// Brief: Setup Arm Error Hold
FUNCTION_BLOCK PUBLIC FB_SetupCtrlError EXTENDS FB_SetupArmCtrlBase
VAR_INPUT
END_VAR
VAR_OUTPUT
END_VAR
VAR
END_VAR

END_FUNCTION_BLOCK

(* stored: Version 1.1.0.1, ProductVersion 3.1.4024.12
   POU FB_SetupCtrlError: Id {1ffb2f4b-fd79-4e75-9d77-eb83ee157467}, SpecialFunc None *)
